Universal Robots PolyScope program: sockets_SeanArnau.urp

Program sockets_SeanArnau (installation=default directory=/programs/Alumnes/Arnau createdIn=5.17.3 lastSavedIn=5.17.3 robotSerialNumber=20205300829)
Calibrated DH parameters: a=[0.000012, -0.242852, -0.179835, 0.000093, -0.000124, 0]; d=[0.151981, 5.088974, 36.181125, -41.139477, 0.085414, 0.092081]; alpha=[1.572112, -0.003585, 0.002783, 1.571586, -1.572466, 0]; deltaTheta=[0, -0.074993, 0.643315, -0.56833, 0.000002, 0]
InitVariablesNode
BeforeStart
  initial_pose := get_actual_tcp_pose()
  ip := "172.23.5.109"
  socket := socket_open(ip, 5858, "s1")
Robot Program (runOnlyOnce=false)
  Loop While (checkContinuously=false) expression=socket≟ False
    socket := socket_open(ip, 5858,"s1")
  Script: socket_send_line(get_actual_tcp_pose(), "s1")
  MoveJ speed 60 deg/s, acceleration 80 deg/s^2 (useActiveTCP=true) feature=Base
    Waypoint Variable (Variable): variable=initial_pose
  read_line := socket_read_ascii_float(6,"s1")
  Loop While (checkContinuously=false) expression=read_line[0]≟0
    read_line := socket_read_ascii_float(6,"s1")
    Wait Sleep waitTime=0.5
  Popup Message (haltProgram=false inputType=Variable) variable=read_line
  posicion := p[read_line[1],read_line[2],read_line[3],read_line[4],read_line[5],read_line[6]]
  MoveJ speed 60 deg/s, acceleration 80 deg/s^2 (useActiveTCP=true) feature=Base
    Waypoint Variable (Variable): variable=posicion
